Staubli VAL3: Deb2304.pgx

program Deb2304()
begin

  dPowerlinkSorti[0]=true

  waitEndMove()
  mov
  movej(ja[0],tstylo,mlent)
  waitEndMove()
  movej(ja[1],tstylo,mlent)
  waitEndMove()
  movej(ja[2],tstylo,mlent)
  waitEndMove()
  movej(ja[3],tstylo,mlent)
  waitEndMove()
  movej(ja[4],tstylo,mlent)
  waitEndMove()
  movej(ja[3],tstylo,mlent)
  waitEndMove()
  movej(ja[2],tstylo,mlent)
  waitEndMove()
  movej(ja[0],tstylo,mlent)
  waitEndMove()

  dPowerlinkSorti[0]=false
end
